{attribute 'qualified_only'}
{attribute 'strict'}
TYPE E_TEST_STATE :
(
	STATE_TEST_OFF				:= 0,
	STATE_TEST_RUNNING
);
END_TYPE

(* stored: Version 1.1.0.1, ProductVersion 3.1.4024.11
   DUT E_TEST_STATE: Id {bf083e7b-1225-46ec-91eb-dd5285cd4b2c} *)
